(* IEC 61131-3 sources: AXOpen/src/_components.cognex.vision/ctrl/src/AxoInsight/v_6_0_0/Tasks, 1 file *)

(* ---- AxoInsightTrigger.st ---- *)
USING AXOpen.Core;
USING AXOpen.Messaging;
USING AXOpen.Messaging.Static;

NAMESPACE AXOpen.Components.Cognex.Vision.v_6_0_0_0
    {S7.extern=ReadWrite}
    CLASS PUBLIC AxoInsightTrigger EXTENDS AXOpen.Core.AxoTask
        VAR PROTECTED
            _progress : INT := 0;
            _infoTimer :  AXOpen.Timers.OnDelayTimer;
            _errorTimer :  AXOpen.Timers.OnDelayTimer;
        END_VAR

        VAR PRIVATE
            _infoTime       :   LTIME := LT#2S;
            _errorTime      :   LTIME := LT#5S;
            _refStatus      :   REF_TO  AxoInsight_Status;
            _refMessenger   :   REF_TO  AxoMessenger;
        END_VAR

        ///<summary>
        /// Runs the logic of this tasks.
        /// >[!IMPORTANT] This method must be called cyclically.
        ///</summary>
        METHOD PUBLIC Run
            VAR_INPUT
                refAcquisitionControl  :   REF_TO  AxoInsight_AcquisitionControl;
                refAcquisitionStatus   :   REF_TO  AxoInsight_AcquisitionStatus;
                refInspectionControl   :   REF_TO  AxoInsight_InspectionControl;
                refInspectionStatus    :   REF_TO  AxoInsight_InspectionStatus;
                refCommandControl      :   REF_TO  AxoInsight_CommandControl;
                refConfig              :   REF_TO  AxoInsight_Config;
                refStatus              :   REF_TO  AxoInsight_Status;
                refResults             :   REF_TO  AxoInsight_Results;
                refInspectionResults   :   REF_TO  AxoInsight_ResultData;
                refResultData          :   REF_TO  ARRAY[*] OF BYTE;
                refMessenger           :   REF_TO  AxoMessenger;
            END_VAR

            VAR
                _index : INT;
                _inspectionCompleted : BOOL;
            END_VAR

            _infoTime := refConfig^.InfoTime;
            _errorTime := refConfig^.ErrorTime;
            _refStatus := refStatus;
            _refMessenger := refMessenger;

            IF THIS.Execute() THEN
                refMessenger^.Serve(THIS);
                IF _progress = 0 THEN
                    refStatus^.Action.Id := UINT#305;
                    refStatus^.Error.Id := UINT#0;
                    refMessenger^.Restore();
                    THIS.CallTimers(FALSE);
                    _progress := _progress + 1;
                END_IF;

                IF _progress = 1 THEN
                    refAcquisitionControl^.TriggerEnable  := TRUE;
                    refAcquisitionControl^.Trigger := FALSE;
                    refAcquisitionControl^.ClearExposureComplete := refAcquisitionStatus^.ExposureComplete;
                    refAcquisitionControl^.SetOffline := FALSE;

                    refInspectionControl^.EnableResultsBuffering := FALSE;
                    refInspectionControl^.AcknowledgeInspectionResults := refInspectionStatus^.ResultsValid;
                    refInspectionControl^.ExtendedUserDataSet := FALSE;
                    refInspectionControl^.ExecuteCommand := FALSE;
                    refInspectionControl^.ClearError := refInspectionStatus^.Error;

                    refCommandControl^.Command:= UINT#0;
                    _progress := _progress + 1;
                END_IF;

                IF _progress = 2 THEN
                    refMessenger^.ActivateOnCondition(ULINT#600, _infoTimer.output, eAxoMessageCategory#Warning);
                    IF _infoTimer.output THEN
                        refStatus^.Error.Id := UINT#600;
                    END_IF;

                    IF NOT refAcquisitionStatus^.ExposureComplete THEN
                        refAcquisitionControl^.ClearExposureComplete := FALSE;
                        THIS.CallTimers(FALSE);
                        _progress := _progress + 1;
                    END_IF;
                END_IF;

                IF _progress = 3 THEN
                    refMessenger^.ActivateOnCondition(ULINT#601, _infoTimer.output, eAxoMessageCategory#Warning);
                    IF _infoTimer.output THEN
                        refStatus^.Error.Id := UINT#601;
                    END_IF;

                    IF NOT refInspectionStatus^.ResultsValid THEN
                        refInspectionControl^.AcknowledgeInspectionResults := FALSE;
                        THIS.CallTimers(FALSE);
                        _progress := _progress + 1;
                    END_IF;
                END_IF;

                IF _progress = 4 THEN
                    refMessenger^.ActivateOnCondition(ULINT#602, _infoTimer.output, eAxoMessageCategory#Warning);
                    IF _infoTimer.output THEN
                        refStatus^.Error.Id := UINT#602;
                    END_IF;

                    IF NOT refInspectionStatus^.Error THEN
                        refInspectionControl^.ClearError := FALSE;
                        THIS.CallTimers(FALSE);
                        _progress := _progress + 1;
                    END_IF;
                END_IF;

                IF _progress = 5 THEN
                    refMessenger^.ActivateOnCondition(ULINT#603, _infoTimer.output, eAxoMessageCategory#Warning);
                    IF _infoTimer.output THEN
                        refStatus^.Error.Id := UINT#603;
                    END_IF;

                    _inspectionCompleted := refInspectionStatus^.InspectionCompleted;
                    IF refAcquisitionStatus^.TriggerReady THEN
                        THIS.CallTimers(FALSE);
                        _progress := _progress + 1;
                    END_IF;
                END_IF;

                IF _progress = 6 THEN
                    refMessenger^.ActivateOnCondition(ULINT#604, _infoTimer.output, eAxoMessageCategory#Warning);
                    IF _infoTimer.output THEN
                        refStatus^.Error.Id := UINT#604;
                    END_IF;

                    refAcquisitionControl^.Trigger := TRUE;
                    IF refAcquisitionStatus^.TriggerAcknowledge THEN
                        THIS.CallTimers(FALSE);
                        _progress := _progress + 1;
                    END_IF;
                END_IF;

                IF _progress = 7 THEN
                    refMessenger^.ActivateOnCondition(ULINT#605, _infoTimer.output, eAxoMessageCategory#Warning);
                    IF _infoTimer.output THEN
                        refStatus^.Error.Id := UINT#605;
                    END_IF;

                    refAcquisitionControl^.Trigger := FALSE;
                    IF _inspectionCompleted <> refInspectionStatus^.InspectionCompleted THEN
                        THIS.CallTimers(FALSE);
                        _progress := _progress + 1;
                    END_IF;
                END_IF;

                IF _progress = 8 THEN
                    refMessenger^.ActivateOnCondition(ULINT#606, _infoTimer.output, eAxoMessageCategory#Warning);
                    IF _infoTimer.output THEN
                        refStatus^.Error.Id := UINT#606;
                    END_IF;

                    IF refInspectionStatus^.ResultsValid THEN
                        THIS.CallTimers(FALSE);
                        _progress := _progress + 1;
                    END_IF;
                END_IF;

                IF _progress = 9 THEN
                    refMessenger^.ActivateOnCondition(ULINT#607, _infoTimer.output, eAxoMessageCategory#Warning);
                    IF _infoTimer.output THEN
                        refStatus^.Error.Id := UINT#607;
                    END_IF;

                    FOR _index := 0 TO (TO_INT(refStatus^.ResultDataSize) - INT#1) DO
                        refInspectionResults^.Data[_index] := refResultData^[_index + 4];
                    END_FOR;
                    FOR _index := refStatus^.ResultDataSize TO 249 DO
                        refInspectionResults^.Data[_index] := BYTE#0;
                    END_FOR;
                    refInspectionResults^.DataChanged := NOT refInspectionResults^.DataChanged ;
                    _progress := _progress + 1;
                END_IF;

                IF _progress = 10 THEN
                    refAcquisitionControl^.Trigger := FALSE;
                    refInspectionControl^.EnableResultsBuffering := FALSE;
                    refInspectionControl^.AcknowledgeInspectionResults := TRUE;
                    THIS.ThrowWhen(refInspectionStatus^.Error);
                    THIS.DoneWhen(TRUE);
                    _progress := 0;
                END_IF;

                THIS.CallTimers(TRUE);

                THIS.ThrowWhen(_errorTimer.output);
            END_IF;
        END_METHOD

        METHOD PRIVATE CallTimers
            VAR_INPUT
                signal : BOOL;
            END_VAR

            _infoTimer.OnDelay(THIS, signal , _infoTime);
            _errorTimer.OnDelay(THIS, signal , _errorTime );
        END_METHOD

        METHOD PROTECTED OVERRIDE OnRestore
            _refStatus^.Action.Id := UINT#309;
            _refStatus^.Error.Id  := UINT#0;
            _refMessenger^.Restore();
            _progress := 0;
            THIS.CallTimers(FALSE);
        END_METHOD

        METHOD PROTECTED OVERRIDE OnAbort
            IF _refStatus <> NULL THEN
                _refStatus^.Action.Id := UINT#601;
            END_IF;
        END_METHOD

        METHOD PROTECTED OVERRIDE OnDone
            IF _refStatus <> NULL THEN
                _refStatus^.Action.Id := UINT#306;
            END_IF;
        END_METHOD

        METHOD PROTECTED OVERRIDE OnError
            IF _refStatus <> NULL THEN
                _refStatus^.Action.Id := UINT#701;
            END_IF;
        END_METHOD

        METHOD PROTECTED OVERRIDE OnStart
            IF _refStatus <> NULL THEN
                _refStatus^.Action.Id := UINT#304;
            END_IF;
        END_METHOD
    END_CLASS
END_NAMESPACE
